FUNCTION_BLOCK ComPort
VAR_INPUT
END_VAR
VAR_OUTPUT
END_VAR
VAR
	(* 	I/O variables for a EL6001 terminal*)
	{attribute 'OPC.UA.DA' := '0'}
	stIn_EL6001 AT %I* : EL6inData22B;	(* linked to the EL6001 in the TwinCAT System Manager *)
	{attribute 'OPC.UA.DA' := '0'}
	stOut_EL6001 AT %Q*	: EL6outData22B;(* linked to the EL6001 in the TwinCAT System Manager *)
	
	(* Internal Variables *) 
	{attribute 'OPC.UA.DA' := '0'}
	fbComPortCtrl : SerialLineControl;
	{attribute 'OPC.UA.DA' := '0'}
	aRxBuffer : ComBuffer;
	{attribute 'OPC.UA.DA' := '0'}
	aTxBuffer : ComBuffer;
	{attribute 'OPC.UA.DA' := '0'}
	bComPortError : BOOL;
	{attribute 'OPC.UA.DA' := '0'}
	eComPortErrorId : ComError_t;

END_VAR

fbComPortCtrl(
	Mode:= SERIALLINEMODE_EL6_22B, 
	pComIn:= ADR(stIn_EL6001), 
	pComOut:= ADR(stOut_EL6001), 
	SizeComIn:= SIZEOF(stIn_EL6001), 
	Error=> , 
	ErrorID=> , 
	TxBuffer:= aTxBuffer, 
	RxBuffer:= aRxBuffer );
IF fbComPortCtrl.Error THEN
	bComPortError := TRUE;
	eComPortErrorId := fbComPortCtrl.ErrorID;
END_IF

PROPERTY PUBLIC ComPortError : BOOL
GET
ComPortError := bComPortError;
END_GET
END_PROPERTY

PROPERTY PUBLIC ComPortErrorId : ComError_t
GET
ComPortErrorId := eComPortErrorId;
END_GET
END_PROPERTY

METHOD PUBLIC Reset
VAR_INPUT
END_VAR
bComPortError := FALSE;
eComPortErrorId := COMERROR_NOERROR;
END_METHOD

PROPERTY PUBLIC RxBuffer : Reference to ComBuffer
GET
RxBuffer REF= aRxBuffer;
END_GET
END_PROPERTY

PROPERTY PUBLIC TxBuffer : Reference to ComBuffer
GET
TxBuffer REF= aTxBuffer;
END_GET
END_PROPERTY

END_FUNCTION_BLOCK

(* stored: Version 1.1.0.1, ProductVersion 3.1.4024.9
   POU ComPort: Id {0e19a445-e458-40ab-ab92-b52b5238a65c}, SpecialFunc None
   Folder Properties: Id {a5dd5c05-7b83-47f5-9305-709e3b555ca9}
   Folder Public: Id {113379e0-29dd-4f31-872b-46cca06cff11}
   Property ComPortError: Id {2b03bf1e-34a6-41b3-8990-4b0ab992219e}
   Get Get: Id {890eeb4c-d359-4ac0-9396-50d500ff2993}
   Property ComPortErrorId: Id {de4acad1-5ae5-4b86-beb8-dee49417e532}
   Get Get: Id {824900ac-1328-4b49-a50e-11ff2ddf2177}
   Method Reset: Id {49bbb285-d2ea-4a40-95de-ee078a347e0d}
   Property RxBuffer: Id {8a5e082e-cbc1-46da-b942-cf233e6f372c}
   Get Get: Id {a17cb106-6bda-4c06-aa94-d27df8cc57e7}
   Property TxBuffer: Id {0fa8534c-1b5c-4ee7-ab13-c983a4934ad0}
   Get Get: Id {d2ec9def-8147-416d-a746-253658f39756} *)
